// TIA Portal V17 export
// export: Created 2022-03-14T09:18:12.6054493Z, ExportSetting WithDefaults, DisplayName Totally Integrated Automation Portal, DisplayVersion V17 Update 2, DisplayName TIA Portal Openness, DisplayVersion V17 Update 2, DisplayName TIA Portal Version Control Interface, DisplayVersion V17, DisplayName STEP 7 Professional, DisplayVersion V17 Update 2, DisplayName STEP 7 Safety, DisplayVersion V17, DisplayName WinCC UA Professional, DisplayVersion V17 Update 2
FUNCTION "FC_1" : Void   // FC1, LAD
{ S7_Optimized_Access := 'TRUE' }
VERSION : 0.1
// stored: AutoNumber true, IsIECCheckEnabled false, SetENOAutomatically false, UDAEnableTagReadback false
   VAR_INPUT
      IN1 : Bool;
      IN2 : Bool;
   END_VAR
   VAR_OUTPUT
      OUT : Bool;
   END_VAR
BEGIN

REGION Network 1
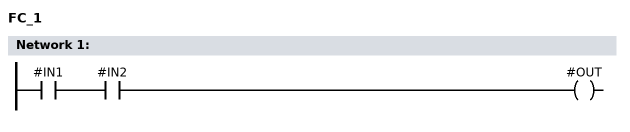
   RUNG wire#powerrail
      Contact( #IN1 )
      Contact( #IN2 )
      Coil( #OUT )
   END_RUNG
   // the same network as SCL:
   #OUT := #IN1 AND #IN2;
END_REGION
END_FUNCTION
